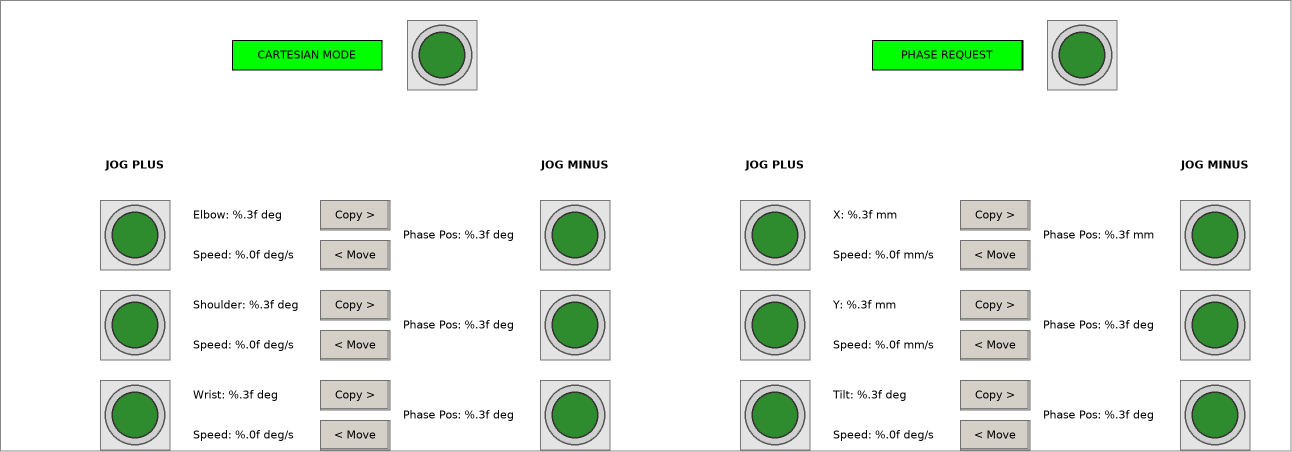
VISUALIZATION CSP_Case_Feed_Kinematic  // 1292x452
    Group (232,20 245x70)
        Rectangle (0,20 150x30), "JOINT MODE", invisible if: csp_case_feed_kinematic.kin_config_cartesian_mode
        PushSwitch (175,0 70x70), variable: csp_case_feed_kinematic.joint_cartesian_mode, input disabled if: csp_case_feed_kinematic.visu_disable_general_command, behaviour: TAP, style: Switch-PushSwitch-Green
        Rectangle (0,20 150x30), "CARTESIAN MODE", invisible if: not csp_case_feed_kinematic.kin_config_cartesian_mode
    Group (872,20 245x70)
        Rectangle (1,20 150x30), "PHASE REQUEST", invisible if: csp_case_feed_kinematic.phase_request
        PushSwitch (175,0 70x70), variable: csp_case_feed_kinematic.phase_request, input disabled if: csp_case_feed_kinematic.visu_disable_phase_request, behaviour: TOGGLE, style: Switch-PushSwitch-Green
        Rectangle (0,20 150x30), "PHASE REQUEST", invisible if: not csp_case_feed_kinematic.phase_request
    Rectangle (60,150 150x30), "JOG PLUS"
    Rectangle (500,150 150x30), "JOG MINUS"
    Group (100,200 510x70)
        Rectangle (90,0 140x30), "Elbow: %.3f deg", text variable: csp_case_feed_kinematic.elbow_actual_position
        PushSwitch (0,0 70x70), variable: csp_case_feed_kinematic.elbow_jog_plus, input disabled if: csp_case_feed_kinematic.visu_disable_ACS_jog_mode, behaviour: TAP, style: Switch-PushSwitch-Green
        PushSwitch (440,0 70x70), variable: csp_case_feed_kinematic.elbow_jog_minus, input disabled if: csp_case_feed_kinematic.visu_disable_ACS_jog_mode, behaviour: TAP, style: Switch-PushSwitch-Green
        Rectangle (90,40 140x30), "Speed: %.0f deg/s", text variable: csp_case_feed_kinematic.elbow_move_speed
            OnMouseDown: write csp_case_feed_kinematic.elbow_move_speed via VisuDialogs.Numpad, min 0, max 100, format %.0f
        Button (220,0 70x30), "Copy >", input disabled if: csp_case_feed_kinematic.visu_disable_ACS_command
            tap csp_case_feed_kinematic.elbow_copy_phase
        Rectangle (300,20 140x30), "Phase Pos: %.3f deg", text variable: csp_case_feed_kinematic.elbow_phase_position
            OnMouseDown: write csp_case_feed_kinematic.elbow_phase_position via VisuDialogs.Numpad, min -200, max 200, format %.3f
        Button (220,40 70x30), "< Move", input disabled if: csp_case_feed_kinematic.visu_disable_ACS_command
            tap csp_case_feed_kinematic.elbow_phase_move
    Group (100,290 510x70)
        Rectangle (90,0 140x30), "Shoulder: %.3f deg", text variable: csp_case_feed_kinematic.shoulder_actual_position
        PushSwitch (0,0 70x70), variable: csp_case_feed_kinematic.shoulder_jog_plus, input disabled if: csp_case_feed_kinematic.visu_disable_ACS_jog_mode, behaviour: TAP, style: Switch-PushSwitch-Green
        PushSwitch (440,0 70x70), variable: csp_case_feed_kinematic.shoulder_jog_minus, input disabled if: csp_case_feed_kinematic.visu_disable_ACS_jog_mode, behaviour: TAP, style: Switch-PushSwitch-Green
        Rectangle (90,40 140x30), "Speed: %.0f deg/s", text variable: csp_case_feed_kinematic.shoulder_move_speed
            OnMouseDown: write csp_case_feed_kinematic.shoulder_move_speed via VisuDialogs.Numpad, min 0, max 100, format %.0f
        Button (220,0 70x30), "Copy >", input disabled if: csp_case_feed_kinematic.visu_disable_ACS_command
            tap csp_case_feed_kinematic.shoulder_copy_phase
        Rectangle (300,20 140x30), "Phase Pos: %.3f deg", text variable: csp_case_feed_kinematic.shoulder_phase_position
            OnMouseDown: write csp_case_feed_kinematic.shoulder_phase_position via VisuDialogs.Numpad, min -200, max 200, format %.3f
        Button (220,40 70x30), "< Move", input disabled if: csp_case_feed_kinematic.visu_disable_ACS_command
            tap csp_case_feed_kinematic.shoulder_phase_move
    Group (100,380 510x70)
        Rectangle (90,0 140x30), "Wrist: %.3f deg", text variable: csp_case_feed_kinematic.wrist_actual_position
        PushSwitch (0,0 70x70), variable: csp_case_feed_kinematic.wrist_jog_plus, input disabled if: csp_case_feed_kinematic.visu_disable_ACS_jog_mode, behaviour: TAP, style: Switch-PushSwitch-Green
        PushSwitch (440,0 70x70), variable: csp_case_feed_kinematic.wrist_jog_minus, input disabled if: csp_case_feed_kinematic.visu_disable_ACS_jog_mode, behaviour: TAP, style: Switch-PushSwitch-Green
        Rectangle (90,40 140x30), "Speed: %.0f deg/s", text variable: csp_case_feed_kinematic.wrist_move_speed
            OnMouseDown: write csp_case_feed_kinematic.wrist_move_speed via VisuDialogs.Numpad, min 0, max 100, format %.0f
        Button (220,0 70x30), "Copy >", input disabled if: csp_case_feed_kinematic.visu_disable_ACS_command
            tap csp_case_feed_kinematic.wrist_copy_phase
        Rectangle (300,20 140x30), "Phase Pos: %.3f deg", text variable: csp_case_feed_kinematic.wrist_phase_position
            OnMouseDown: write csp_case_feed_kinematic.wrist_phase_position via VisuDialogs.Numpad, min -200, max 200, format %.3f
        Button (220,40 70x30), "< Move", input disabled if: csp_case_feed_kinematic.visu_disable_ACS_command
            tap csp_case_feed_kinematic.wrist_phase_move
    Group (740,200 510x70)
        Rectangle (90,0 140x30), "X: %.3f mm", text variable: csp_case_feed_kinematic.x_actual_position
        PushSwitch (0,0 70x70), variable: csp_case_feed_kinematic.x_jog_plus, input disabled if: csp_case_feed_kinematic.visu_disable_MCS_jog_mode, behaviour: TAP, style: Switch-PushSwitch-Green
        PushSwitch (440,0 70x70), variable: csp_case_feed_kinematic.x_jog_minus, input disabled if: csp_case_feed_kinematic.visu_disable_MCS_jog_mode, behaviour: TAP, style: Switch-PushSwitch-Green
        Rectangle (90,40 140x30), "Speed: %.0f mm/s", text variable: csp_case_feed_kinematic.x_move_speed
            OnMouseDown: write csp_case_feed_kinematic.x_move_speed via VisuDialogs.Numpad, min 0, max 100, format %.0f
        Button (220,0 70x30), "Copy >", input disabled if: csp_case_feed_kinematic.visu_disable_MCS_command
            tap csp_case_feed_kinematic.x_copy_phase
        Rectangle (300,20 140x30), "Phase Pos: %.3f mm", text variable: csp_case_feed_kinematic.x_phase_position
            OnMouseDown: write csp_case_feed_kinematic.x_phase_position via VisuDialogs.Numpad, min -2000, max 2000, format %.3f
        Button (220,40 70x30), "< Move", input disabled if: csp_case_feed_kinematic.visu_disable_MCS_command
            tap csp_case_feed_kinematic.x_phase_move
    Rectangle (1140,150 150x30), "JOG MINUS"
    Rectangle (700,150 150x30), "JOG PLUS"
    Group (740,290 510x70)
        Rectangle (90,0 140x30), "Y: %.3f mm", text variable: csp_case_feed_kinematic.y_actual_position
        PushSwitch (0,0 70x70), variable: csp_case_feed_kinematic.y_jog_plus, input disabled if: csp_case_feed_kinematic.visu_disable_MCS_jog_mode, behaviour: TAP, style: Switch-PushSwitch-Green
        PushSwitch (440,0 70x70), variable: csp_case_feed_kinematic.y_jog_minus, input disabled if: csp_case_feed_kinematic.visu_disable_MCS_jog_mode, behaviour: TAP, style: Switch-PushSwitch-Green
        Rectangle (90,40 140x30), "Speed: %.0f mm/s", text variable: csp_case_feed_kinematic.y_move_speed
            OnMouseDown: write csp_case_feed_kinematic.y_move_speed via VisuDialogs.Numpad, min 0, max 100, format %.0f
        Button (220,0 70x30), "Copy >", input disabled if: csp_case_feed_kinematic.visu_disable_MCS_command
            tap csp_case_feed_kinematic.y_copy_phase
        Rectangle (300,20 140x30), "Phase Pos: %.3f deg", text variable: csp_case_feed_kinematic.y_phase_position
            OnMouseDown: write csp_case_feed_kinematic.y_phase_position via VisuDialogs.Numpad, min -100, max 1000, format %.3f
        Button (220,40 70x30), "< Move", input disabled if: csp_case_feed_kinematic.visu_disable_MCS_command
            tap csp_case_feed_kinematic.y_phase_move
    Group (740,380 510x70)
        Rectangle (90,0 140x30), "Tilt: %.3f deg", text variable: csp_case_feed_kinematic.tilt_actual_position
        PushSwitch (0,0 70x70), variable: csp_case_feed_kinematic.tilt_jog_plus, input disabled if: csp_case_feed_kinematic.visu_disable_MCS_jog_mode, behaviour: TAP, style: Switch-PushSwitch-Green
        PushSwitch (440,0 70x70), variable: csp_case_feed_kinematic.tilt_jog_minus, input disabled if: csp_case_feed_kinematic.visu_disable_MCS_jog_mode, behaviour: TAP, style: Switch-PushSwitch-Green
        Rectangle (90,40 140x30), "Speed: %.0f deg/s", text variable: csp_case_feed_kinematic.tilt_move_speed
            OnMouseDown: write csp_case_feed_kinematic.tilt_move_speed via VisuDialogs.Numpad, min 0, max 100, format %.0f
        Button (220,0 70x30), "Copy >", input disabled if: csp_case_feed_kinematic.visu_disable_MCS_command
            tap csp_case_feed_kinematic.tilt_copy_phase
        Rectangle (300,20 140x30), "Phase Pos: %.3f deg", text variable: csp_case_feed_kinematic.tilt_phase_position
            OnMouseDown: write csp_case_feed_kinematic.tilt_phase_position via VisuDialogs.Numpad, min 0, max 150, format %.3f
        Button (220,40 70x30), "< Move", input disabled if: csp_case_feed_kinematic.visu_disable_MCS_command
            tap csp_case_feed_kinematic.tilt_phase_move
END_VISUALIZATION

(* stored: Version 1.1.0.1, ProductVersion 3.1.4024.3
   Visu CSP_Case_Feed_Kinematic: Id {e062a8fe-e97a-4c91-a886-cef712820bd1} *)
